// TIA Portal V17 export
// export: Created 2025-03-10T12:17:41.3737716Z, ExportSetting WithDefaults, DisplayName Totally Integrated Automation Portal, DisplayVersion V17 Update 8, DisplayName TIA Portal Openness, DisplayVersion V17 Update 8, DisplayName TIA Portal Version Control Interface, DisplayVersion V17, DisplayName SINAMICS Startdrive Advanced, DisplayVersion V17 SP2, DisplayName SINAMICS Startdrive G110M, G120, G120C, G120D, G120P, G115D, DisplayVersion V17 SP2, DisplayName SINAMICS Startdrive G130, G150, S120, S150, SINAMICS MV, S210, DisplayVersion V17 SP2, DisplayName STEP 7 Professional, DisplayVersion V17 Update 8, DisplayName SINUMERIK ONE STEP 7 Toolbox, DisplayVersion V17 Update 12, DisplayName SINUMERIK 840D sl STEP 7 Toolbox, DisplayVersion V17 Update 12, DisplayName STEP 7 Safety, DisplayVersion V17 Update 6, DisplayName WinCC Advanced, DisplayVersion V17 Update 8
TYPE "LBP_typeMcp310CPnInput"
TITLE = MCP 310C PN image / Imagen de MCP 310C PN / MCP 310C PN Abbild
// Input image of MCP 310C PN / Imagen de entrada de MCP 310C PN / Eingangsabbild von MCP 310C PN
// stored: IsFailsafeCompliant false
   STRUCT
      standard { S7_SetPoint := 'True'} : "LBP_typeMcp310StandardInput";   // Eingangsabbild von MCP 310 / Input image of MCP 310 / Imagen de entrada de MCP 310
      reserved8 : Byte;
      reserved9 : Byte;
      optionalKey1 : Bool;   // KT-IN1
      optionalKey2 : Bool;   // KT-IN2
      optionalKey3 : Bool;   // KT-IN3
      optionalKey4 : Bool;   // KT-IN4
      optionalKey5 : Bool;   // KT-IN5
      optionalKey6 : Bool;   // KT-IN6
      optionalKey7 : Bool;   // KT-IN7
      optionalKey8 : Bool;   // KT-IN8
      optionalKey9 : Bool;   // KT-IN9
      reserved111 : Bool;
      reserved112 : Bool;
      reserved113 : Bool;
      reserved114 : Bool;
      reserved115 : Bool;
      reserved116 : Bool;
      reserved117 : Bool;
      reserved12 : Byte;
      spindleOvrA : Bool;
      spindleOvrB : Bool;
      spindleOvrC : Bool;
      spindleOvrD : Bool;
      spindleOvrE : Bool;
      reserved135 : Bool;
      reserved136 : Bool;
      reserved137 : Bool;
   END_STRUCT;
END_TYPE
